FUNCTION_BLOCK STRUCT_MUX (* Service Interface Function Block Type *)
  {SET_ATTRIBUTE(GenericClassName, 'GEN_STRUCT_MUX')}
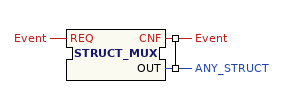
  EVENT_INPUT
    REQ; (* Normal Execution Request *)
  END_EVENT
  EVENT_OUTPUT
    CNF WITH OUT; (* Execution Confirmation *)
  END_EVENT
  VAR_OUTPUT
    OUT : ANY_STRUCT; (* Output *)
  END_VAR
  (* Service APPLICATION/RESOURCE: Service Interface Function Block Type *)
END_FUNCTION_BLOCK
